FUNCTION RefillWater : BOOL
VAR_INPUT
	WaterRefilled		:		BOOL;		// Water is refilled
END_VAR
VAR
END_VAR

// Producing coffee by means of an senseo machine
// Name: Jurriën Arends
// Studentnumer: 515355
// Date: 6-11-2024
// Version: 0.8

// Function: Refill water of coffee machine when it's empty.
IF WaterRefilled = TRUE THEN				// If water is refilled. Waterlevel of reservoir is full. Return variable to 'PrepareMachine'.
  	GVL.WaterLevel := 4;	
  	WaterRefilled:= FALSE;
END_IF;

END_FUNCTION

(* stored: Version 1.1.0.1, ProductVersion 3.1.4024.12
   POU RefillWater: Id {60a29a19-bfa5-4e8c-84ec-0c6eff5f24c7}, SpecialFunc None *)
